// TIA Portal V19 export
DATA_BLOCK "A0303_TraslazioneStrato"   // DB97
// stored: InstanceOfName A0303_TraslazioneStrato_FB, InstanceOfType FB
"A0303_TraslazioneStrato_FB"
   // VAR_INPUT
   //    AreaInterface : "AreaInterface";
   //    ZSI : "udt_ZoneSafetyInterface";
   //    DSI_Feed_Testa : "udt_DeviceSafetyInterface";
   //    DSI_Feed_Coda : "udt_DeviceSafetyInterface";
   //    DSI_Valve : "udt_DeviceSafetyInterface";
   //    DataIn : Struct
   //       OP_Vai_A_Prelievo : Bool;
   //       OP_Prelievo : Bool;
   //       OP_Vai_A_Deposito : Bool;
   //       OP_Deposito : Bool;
   //       LsSensor1 : Bool;
   //       LsSensor2 : Bool;
   //       StratoDepositato_Testa_AnalSens : Int;
   //       StratoDepositato_Coda_AnalSens : Int;
   //    END_STRUCT;
   //    CIn : Struct
   //       SemiAut_Pb { ExternalAccessible := 'False'; ExternalVisible := 'False'; ExternalWritable := 'False'} : Bool;
   //       Manager : Struct
   //          EnableStopDoorOpeningReq : Bool;
   //          EnableStopInPhase : Bool;
   //          EnableStopProgrammed : Bool;
   //          Control_ON : Bool;
   //          CanMoveFreely : Bool;
   //          OP : Struct
   //             VAI_A_PRELIEVO : Bool;
   //             PRELIEVO : Bool;
   //             VAI_A_DEPOSITO : Bool;
   //             DEPOSITO : Bool;
   //          END_STRUCT;
   //       END_STRUCT;
   //       Sollevatore : Struct
   //          OutOfWorkspace : Bool;
   //          ActualPos_Testa : LReal;
   //          ActualPos_Coda : LReal;
   //       END_STRUCT;
   //       Antiribaltamento : Struct
   //          InRestPos : Bool;
   //          InPos0 : Bool;
   //       END_STRUCT;
   //    END_STRUCT;
   //    Config : Struct
   //       Testa : Struct
   //          Ax : "Positioning_EPOS_Machine_Config_NEW";
   //          Manip_Sostegno : "ValveMachine_Config";
   //          Manip_Pareggiatore : "ValveMachine_Config";
   //          SostegnoVrt : "ValveMachine_Config";
   //       END_STRUCT;
   //       Coda : Struct
   //          Ax : "Positioning_EPOS_Machine_Config_NEW";
   //          Manip_Sostegno : "ValveMachine_Config";
   //          Manip_Pareggiatore : "ValveMachine_Config";
   //          SostegnoVrt : "ValveMachine_Config";
   //          DelayMissingCondition { ExternalAccessible := 'False'; ExternalVisible := 'False'; ExternalWritable := 'False'} : Time;
   //       END_STRUCT;
   //       DelayMissingCondition { ExternalAccessible := 'False'; ExternalVisible := 'False'; ExternalWritable := 'False'} : Time;
   //    END_STRUCT;
   // END_VAR
   // VAR_OUTPUT
   //    MachineInterface : "MachineInterface";
   //    COut : Struct
   //       Testa : Struct
   //          Ax : "Positioning_EPOS_Machine_COut";
   //          Manip_Sostegno : "ValveMachine_COut";
   //          Manip_Pareggiatore : "ValveMachine_COut";
   //          SostegnoVrt : "ValveMachine_COut";
   //       END_STRUCT;
   //       Coda : Struct
   //          Ax : "Positioning_EPOS_Machine_COut";
   //          Manip_Sostegno : "ValveMachine_COut";
   //          Manip_Pareggiatore : "ValveMachine_COut";
   //          SostegnoVrt : "ValveMachine_COut";
   //       END_STRUCT;
   //       Cumulativo : Struct
   //          Manip_Sostegno : "ValveMachine_COut";
   //          Manip_Pareggiatore : "ValveMachine_COut";
   //          SostegnoVrt : "ValveMachine_COut";
   //       END_STRUCT;
   //    END_STRUCT;
   // END_VAR
   // VAR_IN_OUT
   //    Par : Struct
   //       Ax_Man : "Positioning_EPOS_Machine_Par";
   //       Ax_Aut : "Mach_Speed_Par";
   //       ToleranceHeight : LReal;
   //       TimeoutTolerance : Time;
   //       Pers_Data_Testa : Struct
   //          EncoderAbsolute_Preset_OK : Bool;
   //          Persistent_ActualPosition : LReal;
   //       END_STRUCT;
   //       Pers_Data_Coda : Struct
   //          EncoderAbsolute_Preset_OK : Bool;
   //          Persistent_ActualPosition : LReal;
   //       END_STRUCT;
   //       Sens_Testa : "Analogic_SensorManagement_Par";
   //       Sens_Coda : "Analogic_SensorManagement_Par";
   //    END_STRUCT;
   //    Par_Mach : Struct
   //       PosPrelievo : LReal;
   //       PosDeposito : LReal;
   //       ToleranceWindow : LReal;
   //    END_STRUCT;
   //    Data_Testa : "Analogic_SensorManagement_Data";
   //    Data_Coda : "Analogic_SensorManagement_Data";
   // END_VAR
   // VAR
   //    Alarm : Struct
   //       Testa : Struct
   //          Ax { S7_SetPoint := 'True'} : "Positioning_EPOS_Machine_Alr";
   //          Manip_Sostegno : "ValveAlr";
   //          Manip_Pareggiatore { S7_SetPoint := 'True'} : "ValveAlr";
   //          SostegnoVrt { S7_SetPoint := 'True'} : "ValveAlr";
   //       END_STRUCT;
   //       Coda : Struct
   //          Ax { S7_SetPoint := 'True'} : "Positioning_EPOS_Machine_Alr";
   //          Manip_Sostegno : "ValveAlr";
   //          Manip_Pareggiatore { S7_SetPoint := 'True'} : "ValveAlr";
   //          SostegnoVrt { S7_SetPoint := 'True'} : "ValveAlr";
   //       END_STRUCT;
   //       StratoDepositatoNoOk : Bool;
   //       CheckBothAxMove : Bool;
   //    END_STRUCT;
   //    Warning : Struct
   //       Testa : Struct
   //          Ax { S7_SetPoint := 'True'} : "Positioning_EPOS_Machine_Wng";
   //          Manip_Sostegno { S7_SetPoint := 'True'} : "ValveMachine_Wng";
   //          Manip_Pareggiatore { S7_SetPoint := 'True'} : "ValveMachine_Wng";
   //          SostegnoVrt { S7_SetPoint := 'True'} : "ValveMachine_Wng";
   //       END_STRUCT;
   //       Coda : Struct
   //          Ax { S7_SetPoint := 'True'} : "Positioning_EPOS_Machine_Wng";
   //          Manip_Sostegno { S7_SetPoint := 'True'} : "ValveMachine_Wng";
   //          Manip_Pareggiatore { S7_SetPoint := 'True'} : "ValveMachine_Wng";
   //          SostegnoVrt { S7_SetPoint := 'True'} : "ValveMachine_Wng";
   //       END_STRUCT;
   //       Sens_Testa { S7_SetPoint := 'True'} : "Analogic_SensorManagement_Warning";
   //       Sens_Coda { S7_SetPoint := 'True'} : "Analogic_SensorManagement_Warning";
   //       MissingCnd : Struct
   //          OP_VAI_A_PRELIEVO : Bool;
   //          OP_PRELIEVO : Bool;
   //          OP_DEPOSITO : Bool;
   //          OP_VAI_A_DEPOSITO : Bool;
   //          SollevatoreInWorkspace : Bool;
   //       END_STRUCT;
   //    END_STRUCT;
   //    HMI : Struct
   //       Selection : Struct
   //          Ax : Int;
   //          Manip_Sostegno : Int;
   //          Manip_Pareggiatore : Int;
   //          SostegnoVrt : Int;
   //       END_STRUCT;
   //       AnalogSensor_Testa : "HMI_Preset";
   //       AnalogSensor_Coda : "HMI_Preset";
   //       Testa : Struct
   //          PbPreset : Bool;
   //          PresetValue : LReal;
   //       END_STRUCT;
   //       Coda : Struct
   //          PbPreset : Bool;
   //          PresetValue : LReal;
   //       END_STRUCT;
   //       AltezzaPaccoTesta : Struct
   //          Target : LReal;
   //          AltezzaMassimaRilevata : LReal;
   //          AltezzaMedia : LReal;
   //          FuoriTolleranza : Bool;
   //       END_STRUCT;
   //       AltezzaPaccoCoda : Struct
   //          Target : LReal;
   //          AltezzaMassimaRilevata : LReal;
   //          AltezzaMedia : LReal;
   //          FuoriTolleranza : Bool;
   //       END_STRUCT;
   //    END_STRUCT;
   //    Sts : Struct
   //       OP_CanMoveFreely : Bool;
   //       OP_Vai_A_Prelievo_Cnd : Bool;
   //       OP_Prelievo_Cnd : Bool;
   //       OP_Deposito_Cnd : Bool;
   //       OP_Vai_A_Deposito_Cnd : Bool;
   //       Coda_PermessoDaSynchOk : Bool;
   //       Testa_PermessoDaSynchOk : Bool;
   //       HeightStackerLayer_Testa : LReal;
   //       HeightStackerLayer_Coda : LReal;
   //       ActPosPhcTesta : LReal;
   //       ActPosPhcCoda : LReal;
   //       MaxHeightDetectedCoda : LReal;
   //       MaxHeightDetectedTesta : LReal;
   //    END_STRUCT;
   //    Ctrl : Struct
   //       Man : Struct
   //          OP_Vai_A_Prelievo : Bool;
   //          OP_Prelievo : Bool;
   //          OP_Deposito : Bool;
   //          OP_Vai_A_Deposito : Bool;
   //       END_STRUCT;
   //       Aut : Struct
   //          OP_Vai_A_Prelievo : Bool;
   //          OP_Prelievo : Bool;
   //          OP_Deposito : Bool;
   //          OP_Vai_A_Deposito : Bool;
   //       END_STRUCT;
   //       OP_Vai_A_Prelievo : Bool;
   //       OP_Prelievo : Bool;
   //       OP_Deposito : Bool;
   //       OP_Vai_A_Deposito : Bool;
   //    END_STRUCT;
   //    Ax_Testa { S7_SetPoint := 'True'} : "Positioning_EPOS_Machine_FB_NEW";
   //    Ax_Coda { S7_SetPoint := 'True'} : "Positioning_EPOS_Machine_FB_NEW";
   //    ValueVelOvr { ExternalAccessible := 'False'; ExternalVisible := 'False'; ExternalWritable := 'False'} : Array[1..10] of Real;
   //    Manip_Sostegno_Testa { S7_SetPoint := 'True'} : "ValveMachine_FB";
   //    Manip_Sostegno_Coda { S7_SetPoint := 'True'} : "ValveMachine_FB";
   //    Manip_Pareggiatore_Testa { S7_SetPoint := 'True'} : "ValveMachine_FB";
   //    Manip_Pareggiatore_Coda { S7_SetPoint := 'True'} : "ValveMachine_FB";
   //    SostegnoVrt_Testa { S7_SetPoint := 'True'} : "ValveMachine_FB";
   //    SostegnoVrt_Coda { S7_SetPoint := 'True'} : "ValveMachine_FB";
   //    StratoDepositato_Testa { S7_SetPoint := 'True'} : "Analogic_SensorManagement";
   //    StratoDepositato_Coda { S7_SetPoint := 'True'} : "Analogic_SensorManagement";
   //    ControlloStrato_Testa : Struct
   //       Enable : Bool;
   //       InsideCheckWindow : Bool;
   //       OutOfTolerance : Bool;
   //    END_STRUCT;
   //    ControlloStrato_Coda : Struct
   //       Enable : Bool;
   //       InsideCheckWindow : Bool;
   //       OutOfTolerance : Bool;
   //    END_STRUCT;
   //    AUX { ExternalAccessible := 'False'; ExternalVisible := 'False'; ExternalWritable := 'False'} : Struct
   //       OP_Vai_A_Prelievo : Bool;
   //       OP_Prelievo : Bool;
   //       OP_Deposito : Bool;
   //       OP_Vai_A_Deposito : Bool;
   //    END_STRUCT;
   //    TON_OP_VAI_A_PRELIEVO_MissingCnd : IEC_TIMER;
   //    TON_OP_VAI_A_DEPOSITO_MissingCnd : IEC_TIMER;
   //    TON_OP_PRELIEVO_MissingCnd : IEC_TIMER;
   //    TON_OP_DEPOSITO_MissingCnd : IEC_TIMER;
   //    TON_StratoDepositatoAlarm { S7_SetPoint := 'True'} : IEC_TIMER;
   //    TON_CheckAxMove { S7_SetPoint := 'True'} : IEC_TIMER;
   //    CheckAxisSynch { S7_SetPoint := 'True'} : "CheckAxisSynch";
   //    BufferHeight { S7_SetPoint := 'True'} : Array[1..9] of LReal;
   // END_VAR
BEGIN
END_DATA_BLOCK
